// TwinCAT 3 PLC project Untitled1
// ProgramVersion: 3.1.4023.0
// libraries:
//   Tc2_Standard, * (Beckhoff Automation GmbH)
//   Tc2_System, * (Beckhoff Automation GmbH)
//   Tc3_Module, * (Beckhoff Automation GmbH)
// project tree:
//   DUTs/ ST_Aligned.TcDUT, ST_AlignedStructs.TcDUT, ST_Packed.TcDUT, U_AlignedStructs.TcDUT
//   / PlcTask.TcTTO
//   POUs/ MAIN.TcPOU
// real-time tasks:
//   TASK PlcTask: cycle T#10ms, priority 20, ADS port 350

CONFIGURATION Untitled1
    RESOURCE PLC ON TwinCAT3
        TASK PlcTask(INTERVAL := T#10ms, PRIORITY := 20);
        PROGRAM MAIN WITH PlcTask : MAIN;
    END_RESOURCE
END_CONFIGURATION

// ---- DUTs/ST_Aligned.TcDUT
{attribute 'pack_mode' := '2'}
TYPE ST_Aligned :						// 14 bytes
STRUCT
	bSwitch		: BOOL		:= FALSE;	// 1 byte
	sText		: STRING[4]	:= 'abcd';	// 5 bytes
	nReal		: REAL		:= 5.845;	// 4 bytes
	nInt		: INT		:= 234;		// 2 bytes
	nByte		: BYTE		:= 76;		// 1 byte
	//nPadding	: BYTE		:= 0;		// 1 byte
END_STRUCT
END_TYPE

// ---- DUTs/ST_AlignedStructs.TcDUT
TYPE ST_AlignedStructs :
STRUCT
	stAligned1	: ST_Aligned;
	stAligned2	: ST_Aligned;
	stAligned3	: ST_Aligned;
END_STRUCT
END_TYPE

// ---- DUTs/ST_Packed.TcDUT
{attribute 'pack_mode' := '1'}
TYPE ST_Packed :					// 13 bytes
STRUCT
	bSwitch	: BOOL		:= FALSE;	// 1 byte
	sText	: STRING[4]	:= 'abcd';	// 5 bytes
	nReal	: REAL		:= 5.845;	// 4 bytes
	nInt	: INT		:= 234;		// 2 bytes
	nByte	: BYTE		:= 76;		// 1 byte
END_STRUCT
END_TYPE

// ---- DUTs/U_AlignedStructs.TcDUT
TYPE U_AlignedStructs :
UNION
	aAlignedStructs		: ARRAY[0..2] OF ST_Aligned;
	stAlignedStructs	: ST_AlignedStructs;
END_UNION
END_TYPE

// ---- POUs/MAIN.TcPOU
PROGRAM MAIN
VAR
	byByte		AT %MB0	: ARRAY[0..1027] OF BYTE;
	i					: INT;
	moreBytes			: ARRAY[0..8192] OF BYTE;
	stInput				: ST_Packed;
	stOutput			: ST_Packed;
	stAlignedInput		: ST_Aligned;
	stAlignedOutput		: ST_Aligned;
	uAlignedInput		: U_AlignedStructs;
	uAlignedOutput		: U_AlignedStructs;
END_VAR

FOR i := 4 TO 1027 BY 1 DO
	byByte[i] := byByte[i] + 1;
END_FOR
stOutput := stInput;
stAlignedOutput := stAlignedInput;
uAlignedOutput.aAlignedStructs := uAlignedInput.aAlignedStructs;

END_PROGRAM
